TYPE ST_AxisError:
STRUCT
//PLCopen function block errors
    nPowerErrorID: UDINT;
    nMoveAbsoluteErrorID: UDINT;
	nLocalMoveAbsoluteErrorID: UDINT;
    nMoveRelativeErrorID: UDINT;
	nLocalMoveRelativeErrorID: UDINT;
    nMoveVelocityErrorID: UDINT;
	nLocalMoveVelocityErrorID: UDINT;
    nMoveModuloErrorID: UDINT;
    nJogErrorID: UDINT;
    nHomeErrorID: UDINT;
    nHaltErrorID: UDINT;
    nResetErrorID: UDINT;
    nStopErrorID: UDINT;
    nGearInMultiMasterErrorID: UDINT;
    nGearOutErrorID: UDINT;
	nSetPositionErrorID : UDINT;
    fbWriteParameterErrorId: UDINT;
    fbReadParameterErrorId: UDINT;
//Error from the NC
    nNCErrorID : UDINT;
END_STRUCT
END_TYPE

(* stored: Version 1.1.0.1, ProductVersion 3.1.4026.18
   DUT ST_AxisError: Id {b605e536-99a4-4241-8b01-b55c227dfd1d} *)
